SUBAPPLICATION Uebung_014_AXb (* Container (visible/invisible) *)
  (* Standard: 61499-2; Description: Copyright (c) 2023 Meisterschulen am Ostbahnhof This program and the accompanying materials are made available under the terms of the Eclipse Public License 2.0 which is available at https://www.eclipse.org/legal/epl-2.0/ SPDX-License-Identifier: EPL-2.0 *)
  (* Version 1.0, 2023-10-23, Franz Höpfinger, Meisterschulen am Ostbahnhof, initial API and implementation and/or initial documentation *)
  PACKAGE Uebungen;
  IMPORT Uebungen::const::UT::DefaultPool::Container_B;
  IMPORT Uebungen::const::UT::DefaultPool::SoftKey_F1;
  IMPORT Uebungen::const::UT::DefaultPool::SoftKey_F2;
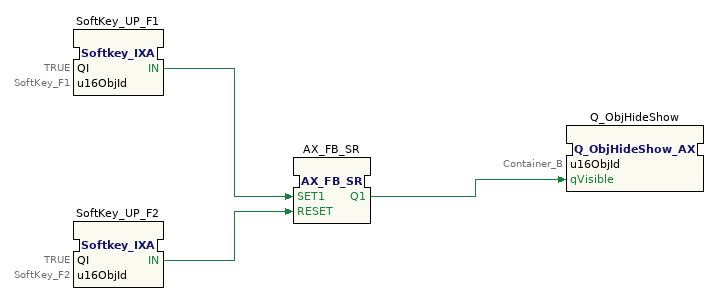
  FBS
    SoftKey_UP_F1 : isobus::UT::io::Softkey::Softkey_IXA(QI := TRUE, u16ObjId := SoftKey_F1);
    SoftKey_UP_F2 : isobus::UT::io::Softkey::Softkey_IXA(QI := TRUE, u16ObjId := SoftKey_F2);
    AX_FB_SR : adapter::iec61131::bistableElements::AX_FB_SR;
    Q_ObjHideShow : isobus::UT::Q::Q_ObjHideShow_AX(u16ObjId := Container_B);
  END_FBS
  ADAPTER_CONNECTIONS
    AX_FB_SR.Q1 TO Q_ObjHideShow.qVisible;
    SoftKey_UP_F1.IN TO AX_FB_SR.SET1;
    SoftKey_UP_F2.IN TO AX_FB_SR.RESET;
  END_CONNECTIONS
END_SUBAPPLICATION
